PROGRAM P_Sensor_Handling
VAR
END_VAR


// Magneettisensorit: SM
//		Kierrosluku, gato/perron ohitus
//		Luukku/ovi johonkin ja varmistamaan että se on kiinni

// Lämpösensori
//		Boxin sisällä, mittaa ympäristön lämpötilaa
//		Derivoidaan ja analogitulosta luodaan ihmelukuja ja graafeja HMI:hin

// Valosensori
//		Gato/perron ohitus maaliviivalla

END_PROGRAM

(* stored: Version 1.1.0.1, ProductVersion 3.1.4024.10
   POU P_Sensor_Handling: Id {ff981f03-5d81-4652-8271-95efea1a58f8}, SpecialFunc None *)
